INTERFACE ITcoCoordinator

METHOD MoveNext : BOOL
END_METHOD

METHOD Retry : BOOL
VAR_INPUT
	inFromState : INT;
END_VAR
END_METHOD

METHOD Terminate : BOOL
END_METHOD

END_INTERFACE

(* stored: Version 1.1.0.1
   Itf ITcoCoordinator: Id {7e9d8dd7-8258-0db9-2f48-d239f9350708}
   Method MoveNext: Id {cb4af035-e41b-0478-18b7-dacf0755afa8}
   Method Retry: Id {8d8f4ae5-b94a-0914-01c6-6cb6d5246300}
   Method Terminate: Id {07bad117-907a-0eee-1668-f0c7019a392a} *)
